(* PLC project CoDeSys External Library Template, WAGO e!COCKPIT e!COCKPIT, author 3S - Smart Software Solutions GmbH *)
(* stored: creationDateTime 2019-10-29T12:37:19.4177669, version 3.5.5.30, modificationDateTime 2019-10-29T12:36:39.3744516, organization 3S - Smart Software Solutions GmbH *)
(* Library project template with all possible element types, docu and a sample project structure *)

(* values of enumPPPSPomieszczenie: SalaLekcyjna: Sale lekcyjne, przedszkolne, świetlica, biblioteka (20 st. C); SalaNiemowlat: Sale niemowląt, dziecięce w żłobkach (24 st. C); Rehabilitacyjne: Pomieszczenia rehabilitacyjne SPON (24 st. C); Korytarz: Korytarze (20 st. C); Szatnia: Szatnie (16 st. C); SalaGimnastyczna: Sale gimnastyczne (16 st. C); Lazienka: Łazienki i ustępy (24 st. C); PomieszczenieBiurowe: Pomieszczenia biurowe i administracyjne (20 st. C); PomieszczenieMieszkalne: Pomieszczenia mieszkalne, przedpokoje, kuchnie (20 st. C); Magazyn: Pomieszczenia magazynowe (16 st. C) *)

(* Autor: Artur Wyszomirski, 2018-10-15-AW; Prawa majątkowe: Solwena Sp. z o.o., Aktualizacje: Opis: enum służy do obsługi rodzajów pomieszczeń w budynkach PPP Sopot (ENGIE) *)
{attribute 'qualified_only'}
{attribute 'strict'}
TYPE enumPPPSPomieszczenie : (SalaLekcyjna := 0, SalaNiemowlat := 1, Rehabilitacyjne := 2, Korytarz := 3, Szatnia := 4, SalaGimnastyczna := 5, Lazienka := 6, PomieszczenieBiurowe := 7, PomieszczenieMieszkalne := 8, Magazyn := 9);
END_TYPE
